// TIA Portal V17 export
// export: Created 2023-12-05T13:40:22.4546774Z, ExportSetting WithDefaults, DisplayName Totally Integrated Automation Portal, DisplayVersion V17, DisplayName TIA Portal Openness, DisplayVersion V17, DisplayName TIA Portal Version Control Interface, DisplayVersion V17, DisplayName SINAMICS Startdrive Advanced, DisplayVersion V17, DisplayName SINAMICS Startdrive G130, G150, S120, S150, SINAMICS MV, S210, DisplayVersion V17, DisplayName SINAMICS Startdrive G110M, G120, G120C, G120D, G120P, G115D, DisplayVersion V17, DisplayName STEP 7 Professional, DisplayVersion V17, DisplayName STEP 7 Safety, DisplayVersion V17, DisplayName WinCC Professional, DisplayVersion V17
FUNCTION "FC530 CPW_V5_1_7 Alarms" : Void   // FC530, LAD
{ S7_Optimized_Access := 'TRUE' }
VERSION : 0.1
// LG 30.06.2022 => Structured in block changed to CPW V5.1.7
// RB 14.09.2021 => Block adapted to SB CPW_V5_1_6
// 3.06 => split alarms for Ack and no Ack display
// 7.05 => block modyfied to work with CPW V5_1_0 IDB data
// stored: AutoNumber false, IsIECCheckEnabled false, SetENOAutomatically false, UDAEnableTagReadback false
   VAR_INPUT
      AckStep : Bool;
      "SB DB" : Int;
      "Alarm DB" : Int;
      "Alarm Offset" : Int;
   END_VAR
   VAR_TEMP
      "SB DBW" : Word;
      "AL DBW" : Word;
      "TR DBW" : Word;
   END_VAR
BEGIN

NETWORK
TITLE = Initialization
      L     #"SB DB";
      T     #"SB DBW";
      L     #"Alarm DB";
      T     #"AL DBW";
      L     #"Alarm Offset";
      SLD   3;
      LAR1;

NETWORK
TITLE = Faults
      CLR;
      OPN   DB [#"SB DBW"];
      L     %DBW156;
      OPN   DB [#"AL DBW"];
      T     DBW [AR1, P#0.0];

      OPN   DB [#"SB DBW"];
      L     %DBW158;
      OPN   DB [#"AL DBW"];
      T     DBW [AR1, P#2.0];

      CLR;
      OPN   DB [#"SB DBW"];
      A     %DBX166.6;
      OPN   DB [#"AL DBW"];
      =     DBX [AR1, P#10.6];

      CLR;
      OPN   DB [#"SB DBW"];
      A     %DBX166.7;
      OPN   DB [#"AL DBW"];
      =     DBX [AR1, P#10.7];

      CLR;
      OPN   DB [#"SB DBW"];
      A     %DBX167.0;
      OPN   DB [#"AL DBW"];
      =     DBX [AR1, P#11.0];

      CLR;
      OPN   DB [#"SB DBW"];
      A     %DBX167.1;
      OPN   DB [#"AL DBW"];
      =     DBX [AR1, P#11.1];

      CLR;
      OPN   DB [#"SB DBW"];
      A     %DBX167.2;
      OPN   DB [#"AL DBW"];
      =     DBX [AR1, P#11.2];

      CLR;
      OPN   DB [#"SB DBW"];
      A     %DBX167.3;
      OPN   DB [#"AL DBW"];
      =     DBX [AR1, P#11.3];

      OPN   DB [#"SB DBW"];
      L     %DBB174;
      OPN   DB [#"AL DBW"];
      T     DBB [AR1, P#18.0];

      CLR;
      OPN   DB [#"SB DBW"];
      A     %DBX175.0;
      OPN   DB [#"AL DBW"];
      =     DBX [AR1, P#19.0];



NETWORK
TITLE = Faults Acknowledge step
      A     #AckStep;
      JCN   en1;

      CLR;
      OPN   DB [#"SB DBW"];
      L     %DBW164;
      OPN   DB [#"AL DBW"];
      T     DBW [AR1, P#8.0];

      OPN   DB [#"SB DBW"];
      A     %DBX166.0;
      OPN   DB [#"AL DBW"];
      =     DBX [AR1, P#10.0];

      OPN   DB [#"SB DBW"];
      A     %DBX166.4;
      OPN   DB [#"AL DBW"];
      =     DBX [AR1, P#10.4];

      OPN   DB [#"SB DBW"];
      A     %DBX166.5;
      OPN   DB [#"AL DBW"];
      =     DBX [AR1, P#10.5];

      OPN   DB [#"SB DBW"];
      A     %DBX167.4;
      OPN   DB [#"AL DBW"];
      =     DBX [AR1, P#11.4];

      OPN   DB [#"SB DBW"];
      A     %DBX167.5;
      OPN   DB [#"AL DBW"];
      =     DBX [AR1, P#11.5];

      OPN   DB [#"SB DBW"];
      A     %DBX167.6;
      OPN   DB [#"AL DBW"];
      =     DBX [AR1, P#11.6];

      CLR;
      OPN   DB [#"SB DBW"];
      L     %DBW168;
      OPN   DB [#"AL DBW"];
      T     DBW [AR1, P#12.0];

      CLR;
      OPN   DB [#"SB DBW"];
      L     %DBW170;
      OPN   DB [#"AL DBW"];
      T     DBW [AR1, P#14.0];

      CLR;
      OPN   DB [#"SB DBW"];
      L     %DBB172;
      OPN   DB [#"AL DBW"];
      T     DBB [AR1, P#16.0];


      OPN   DB [#"SB DBW"];
      A     %DBX173.0;
      OPN   DB [#"AL DBW"];
      =     DBX [AR1, P#17.0];

      OPN   DB [#"SB DBW"];
      A     %DBX173.1;
      OPN   DB [#"AL DBW"];
      =     DBX [AR1, P#17.1];

      OPN   DB [#"SB DBW"];
      A     %DBX173.2;
      OPN   DB [#"AL DBW"];
      =     DBX [AR1, P#17.2];

      OPN   DB [#"SB DBW"];
      A     %DBX175.1;
      OPN   DB [#"AL DBW"];
      =     DBX [AR1, P#19.1];

      OPN   DB [#"SB DBW"];
      A     %DBX175.2;
      OPN   DB [#"AL DBW"];
      =     DBX [AR1, P#19.2];

      OPN   DB [#"SB DBW"];
      A     %DBX175.3;
      OPN   DB [#"AL DBW"];
      =     DBX [AR1, P#19.3];

      OPN   DB [#"SB DBW"];
      A     %DBX175.4;
      OPN   DB [#"AL DBW"];
      =     DBX [AR1, P#19.4];


en1:  NOP   0;
END_FUNCTION
